INTERFACE I_InfeedModule

PROPERTY CfgInfeed : REFERENCE TO ST_InfeedConfig
GET
END_GET
END_PROPERTY

PROPERTY CmdInfeed : REFERENCE TO ST_InfeedCommand
GET
END_GET
END_PROPERTY

PROPERTY RcpInfeed : REFERENCE TO ST_InfeedRecipe
GET
END_GET
END_PROPERTY

PROPERTY StsInfeed : REFERENCE TO ST_InfeedStatus
GET
END_GET
END_PROPERTY

END_INTERFACE

(* stored: Version 1.1.0.1, ProductVersion 3.1.4024.12
   Itf I_InfeedModule: Id {84b9f046-0100-4599-8408-578c34a575cb}
   Property CfgInfeed: Id {b29931a9-9817-474e-8ca1-59c1457c649f}
   Get Get: Id {e0d3fd3e-6654-4bfd-853b-eee5bea719ce}
   Property CmdInfeed: Id {e6301070-c211-41ad-81f3-4480d50714a9}
   Get Get: Id {f9e36858-40ee-4236-be6e-fcf9fe92ad12}
   Property RcpInfeed: Id {634fabee-b302-4ec9-9dd0-33bdc60c8e4f}
   Get Get: Id {779326bf-a771-4f91-a78d-e6249f69505d}
   Property StsInfeed: Id {e288481d-1160-4ae0-940d-42a0dbe603a6}
   Get Get: Id {0e99212c-9f64-47c8-986f-b9dd2f46ed97} *)
